FUNCTION_BLOCK XY_VIEWL (* Two-Dimensional Mechanism View with Local Data Publish/Subscribe *)
  (* Standard: IEC 61499; Classification: View; ApplicationDomain: Material Handling; Function: Two-axis motion *)
  (* Version 0.0, 2006-06-22, JHC, Holobloc Inc, Derived from MECHC_VIEWL for XY_VIEW. *)
  (* Compiler header: package fb.rt.mva; import fb.rt.net.*; *)
  (* Compiler classdef: public class XY_VIEWL extends FBMVCD *)
  (* Compiler Java Sun JDK 1.5.0 *)
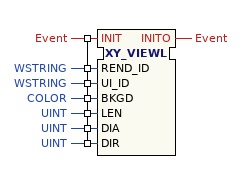
  EVENT_INPUT
    INIT WITH REND_ID, UI_ID, BKGD, LEN, DIA, DIR; (* Initialize *)
  END_EVENT
  EVENT_OUTPUT
    INITO; (* Initialized *)
  END_EVENT
  VAR_INPUT
    REND_ID : WSTRING; (* Rendering Data Channel from Model *)
    UI_ID : WSTRING; (* User Input Channel to Model *)
    BKGD : COLOR := blue; (* Background Color *)
    LEN : UINT; (* Length in Diameters *)
    DIA : UINT; (* Diameter *)
    DIR : UINT; (* Orientation:0=L/R,1=T/B,2=R/L,3=B/T *)
  END_VAR
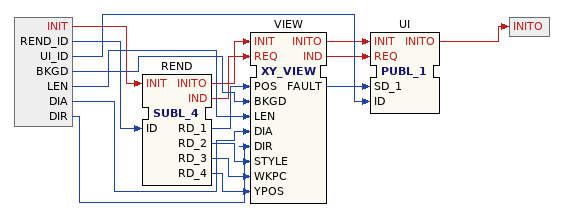
  FBS
    REND : SUBL_4;
    VIEW : XY_VIEW;
    UI : PUBL_1;
  END_FBS
  EVENT_CONNECTIONS
    INIT TO REND.INIT;
    REND.INITO TO VIEW.INIT;
    VIEW.INITO TO UI.INIT;
    UI.INITO TO INITO;
    REND.IND TO VIEW.REQ;
    VIEW.IND TO UI.REQ;
  END_CONNECTIONS
  DATA_CONNECTIONS
    REND.RD_1 TO VIEW.POS;
    VIEW.FAULT TO UI.SD_1;
    REND_ID TO REND.ID;
    UI_ID TO UI.ID;
    BKGD TO VIEW.BKGD;
    LEN TO VIEW.LEN;
    DIA TO VIEW.DIA;
    DIR TO VIEW.DIR;
    REND.RD_2 TO VIEW.STYLE;
    REND.RD_3 TO VIEW.WKPC;
    REND.RD_4 TO VIEW.YPOS;
  END_CONNECTIONS
END_FUNCTION_BLOCK
